Omron CX-Programmer project NuevoProyecto (CX-Programmer 9.61)

# PLC TunelDosTrenes: CJ2M CPU11

## Program NuevoPrograma1 (cyclic task 0)
Local symbols
Aproximación1 0.12 BOOL  ; 0.12
Aproximación2 0.14 BOOL  ; 0.14
P0 2.00 BOOL
P1 2.01 BOOL
P2 2.02 BOOL
P3 2.03 BOOL
Rojo1 1.08 BOOL  ; 1.08
Rojo2 1.09 BOOL  ; 1.09
Salida1 0.13 BOOL  ; 0.13
Salida2 0.15 BOOL  ; 0.15
Verde1 1.00 BOOL  ; 1.00
Verde2 1.01 BOOL  ; 1.01

### Section main

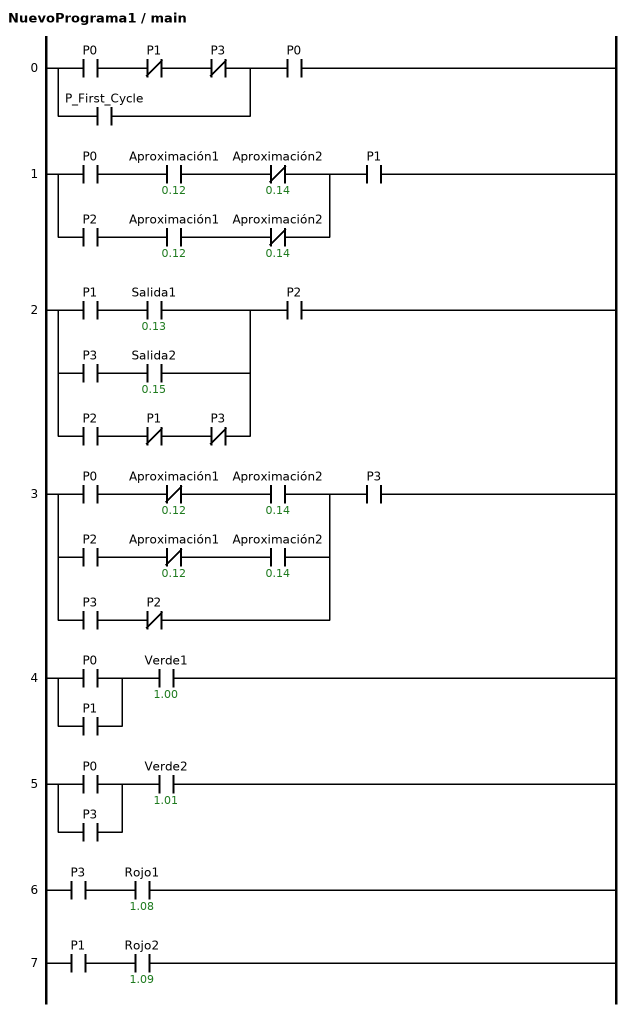
; rung 0
LD P0
ANDNOT P1
ANDNOT P3
OR P_First_Cycle
AND P0
; rung 1
LD P0
AND Aproximación1  ; 0.12
ANDNOT Aproximación2  ; 0.14
LD P2
AND Aproximación1  ; 0.12
ANDNOT Aproximación2  ; 0.14
ORLD
AND P1
; rung 2
LD P1
AND Salida1  ; 0.13
LD P3
AND Salida2  ; 0.15
ORLD
LD P2
ANDNOT P1
ANDNOT P3
ORLD
AND P2
; rung 3
LD P0
ANDNOT Aproximación1  ; 0.12
AND Aproximación2  ; 0.14
LD P2
ANDNOT Aproximación1  ; 0.12
AND Aproximación2  ; 0.14
ORLD
LD P3
ANDNOT P2
ORLD
AND P3
; rung 4
LD P0
OR P1
AND Verde1  ; 1.00
; rung 5
LD P0
OR P3
AND Verde2  ; 1.01
; rung 6
LD P3
AND Rojo1  ; 1.08
; rung 7
LD P1
AND Rojo2  ; 1.09

### Section END
; rung 0
END(001)